// Mitsubishi GX Works2 project: Real Project Capstone   PLC: FX3U/FX3UC

PROGRAM MAIN
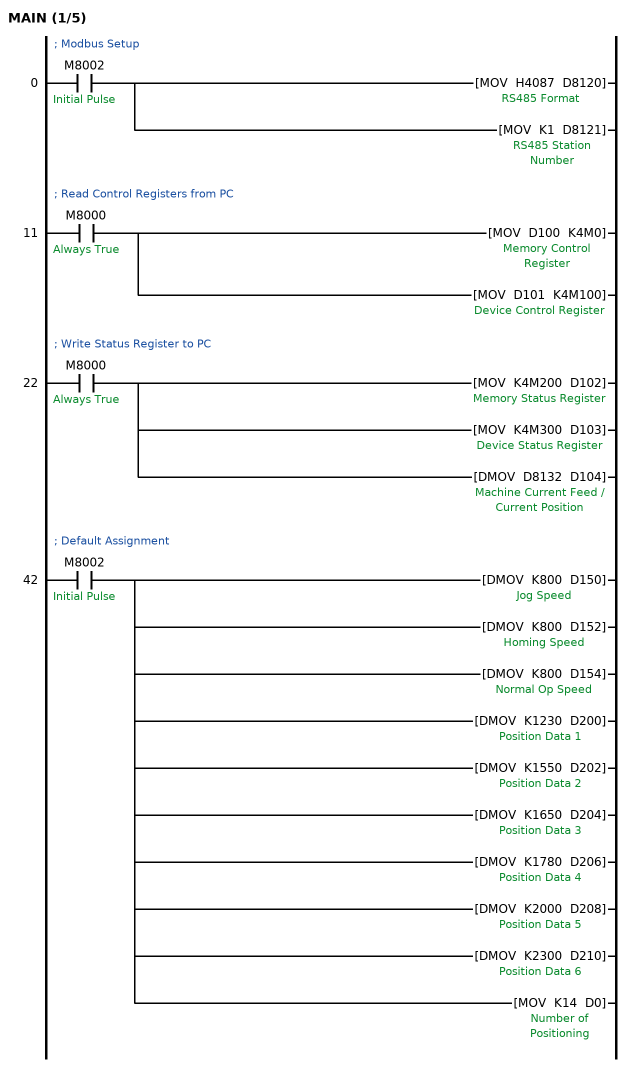
; Modbus Setup
0     LD      M8002  ; Initial Pulse
      MOV     H4087 D8120  ; RS485 Format
      MOV     K1 D8121  ; RS485 Station Number
; Read Control Registers from PC
11    LD      M8000  ; Always True
      MOV     D100 K4M0  ; Memory Control Register / Auto/Man Control
      MOV     D101 K4M100  ; Device Control Register / Light Control
; Write Status Register to PC
22    LD      M8000  ; Always True
      MOV     K4M200 D102  ; Start/Stop Status / Memory Status Register
      MOV     K4M300 D103  ; Light Status / Device Status Register
      DMOV    D8132 D104  ; Machine Current Feed / Current Position
; Default Assignment
42    LD      M8002  ; Initial Pulse
      DMOV    K800 D150  ; Jog Speed
      DMOV    K800 D152  ; Homing Speed
      DMOV    K800 D154  ; Normal Op Speed
      DMOV    K1230 D200  ; Position Data 1
      DMOV    K1550 D202  ; Position Data 2
      DMOV    K1650 D204  ; Position Data 3
      DMOV    K1780 D206  ; Position Data 4
      DMOV    K2000 D208  ; Position Data 5
      DMOV    K2300 D210  ; Position Data 6
      MOV     K14 D0  ; Number of Positioning
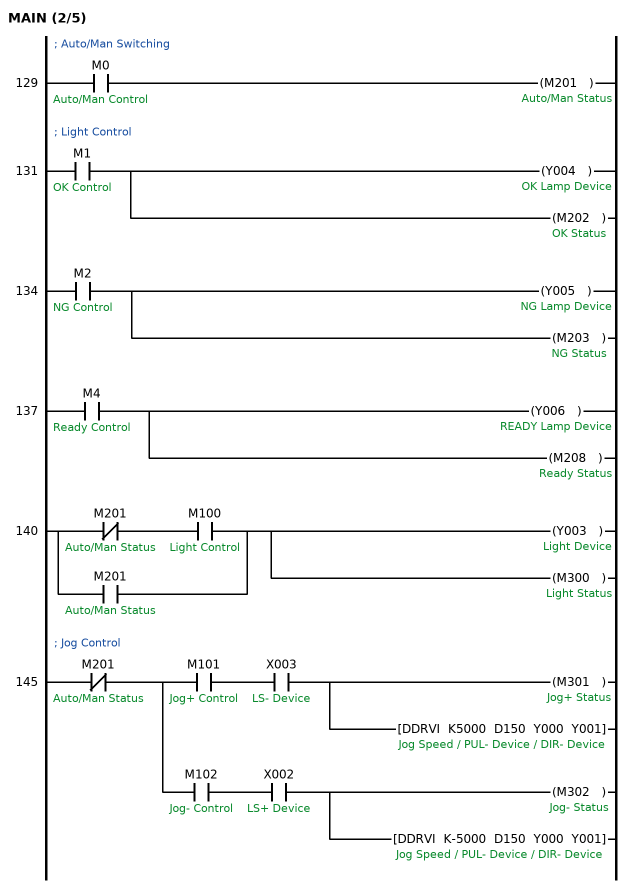
; Auto/Man Switching
129   LD      M0  ; Auto/Man Control
      OUT     M201  ; Auto/Man Status
; Light Control
131   LD      M1  ; OK Control
      OUT     Y004  ; OK Lamp Device
      OUT     M202  ; OK Status
134   LD      M2  ; NG Control
      OUT     Y005  ; NG Lamp Device
      OUT     M203  ; NG Status
137   LD      M4  ; Ready Control
      OUT     Y006  ; READY Lamp Device
      OUT     M208  ; Ready Status
140   LDI     M201  ; Auto/Man Status
      AND     M100  ; Light Control
      OR      M201  ; Auto/Man Status
      OUT     Y003  ; Light Device
      OUT     M300  ; Light Status
; Jog Control
145   LDI     M201  ; Auto/Man Status
      MPS
      AND     M101  ; Jog+ Control
      AND     X003  ; LS- Device
      OUT     M301  ; Jog+ Status
      DDRVI   K5000 D150 Y000 Y001  ; PUL- Device / DIR- Device
      MPP
      AND     M102  ; Jog- Control
      AND     X002  ; LS+ Device
      OUT     M302  ; Jog- Status
      DDRVI   K-5000 D150 Y000 Y001
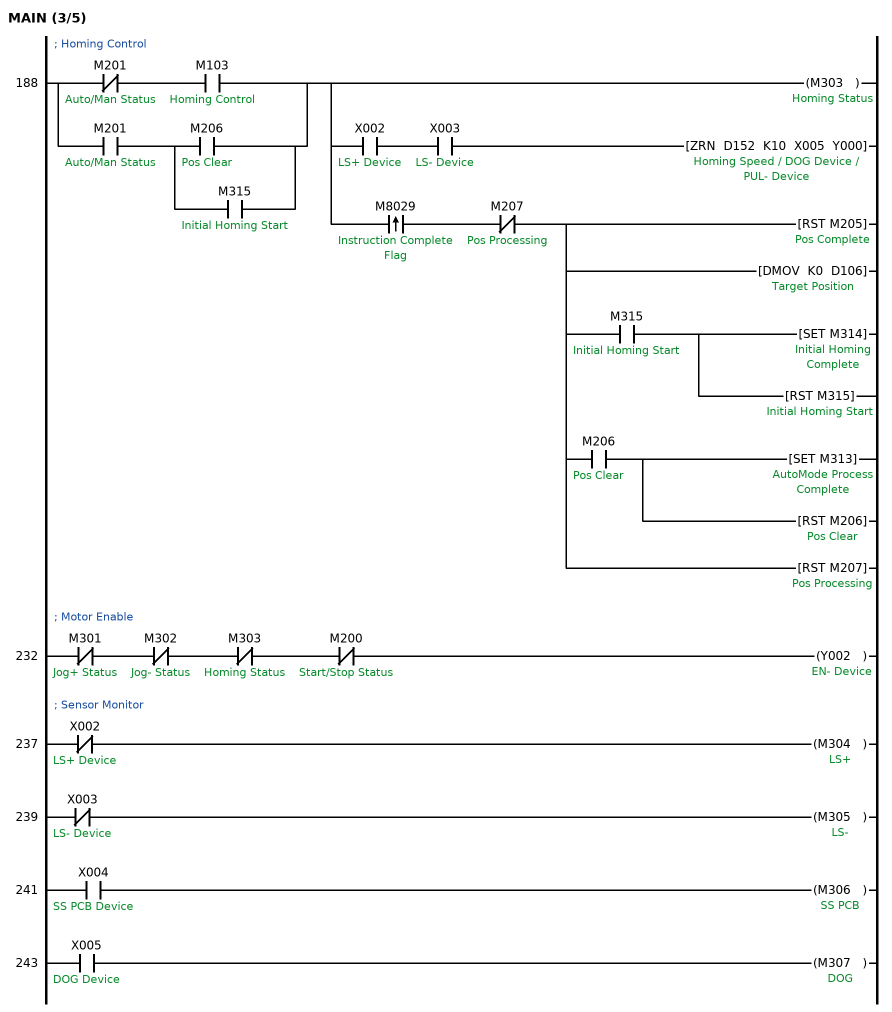
; Homing Control
188   LDI     M201  ; Auto/Man Status
      AND     M103  ; Homing Control
      LD      M201  ; Auto/Man Status
      LD      M206  ; Pos Clear
      OR      M315  ; Initial Homing Start
      ANB
      ORB
      OUT     M303  ; Homing Status
      MPS
      AND     X002  ; LS+ Device
      AND     X003  ; LS- Device
      ZRN     D152 K10 X005 Y000  ; DOG Device
      MPP
      ANDP    M8029  ; Instruction Complete Flag
      ANI     M207  ; Pos Processing
      RST     M205  ; Pos Complete
      DMOV    K0 D106  ; Target Position
      MPS
      AND     M315  ; Initial Homing Start
      SET     M314  ; Initial Homing Complete
      RST     M315  ; Initial Homing Start
      MRD
      AND     M206  ; Pos Clear
      SET     M313  ; AutoMode Process Complete
      RST     M206  ; Pos Clear
      MPP
      RST     M207  ; Pos Processing
; Motor Enable
232   LDI     M301  ; Jog+ Status
      ANI     M302  ; Jog- Status
      ANI     M303  ; Homing Status
      ANI     M200  ; Start/Stop Status
      OUT     Y002  ; EN- Device
; Sensor Monitor
237   LDI     X002  ; LS+ Device
      OUT     M304  ; LS+
239   LDI     X003  ; LS- Device
      OUT     M305  ; LS-
241   LD      X004  ; SS PCB Device
      OUT     M306  ; SS PCB
243   LD      X005  ; DOG Device
      OUT     M307  ; DOG
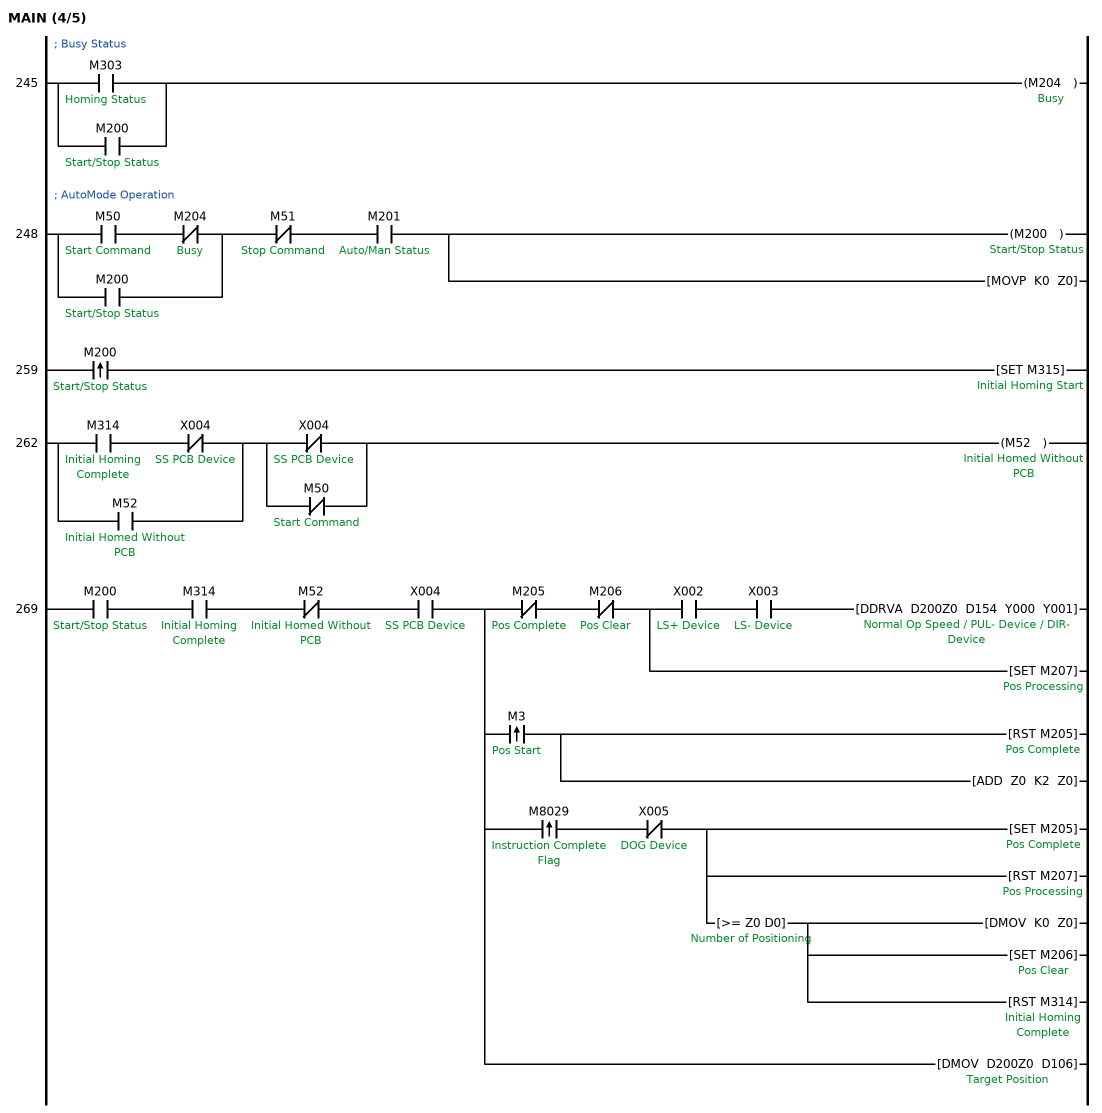
; Busy Status
245   LD      M303  ; Homing Status
      OR      M200  ; Start/Stop Status
      OUT     M204  ; Busy
; AutoMode Operation
248   LD      M50  ; Start Command
      ANI     M204  ; Busy
      OR      M200  ; Start/Stop Status
      ANI     M51  ; Stop Command
      AND     M201  ; Auto/Man Status
      OUT     M200  ; Start/Stop Status
      MOVP    K0 Z0
259   LDP     M200  ; Start/Stop Status
      SET     M315  ; Initial Homing Start
262   LD      M314  ; Initial Homing Complete
      ANI     X004  ; SS PCB Device
      OR      M52  ; Initial Homed Without PCB
      LDI     X004  ; SS PCB Device
      ORI     M50  ; Start Command
      ANB
      OUT     M52  ; Initial Homed Without PCB
269   LD      M200  ; Start/Stop Status
      AND     M314  ; Initial Homing Complete
      ANI     M52  ; Initial Homed Without PCB
      AND     X004  ; SS PCB Device
      MPS
      ANI     M205  ; Pos Complete
      ANI     M206  ; Pos Clear
      MPS
      AND     X002  ; LS+ Device
      AND     X003  ; LS- Device
      DDRVA   D200Z0 D154 Y000 Y001
      MPP
      SET     M207  ; Pos Processing
      MRD
      ANDP    M3  ; Pos Start
      RST     M205  ; Pos Complete
      ADD     Z0 K2 Z0
      MRD
      ANDP    M8029  ; Instruction Complete Flag
      ANI     X005  ; DOG Device
      SET     M205  ; Pos Complete
      RST     M207  ; Pos Processing
      AND>=   Z0 D0  ; Number of Positioning
      DMOV    K0 Z0
      SET     M206  ; Pos Clear
      RST     M314  ; Initial Homing Complete
      MPP
      DMOV    D200Z0 D106
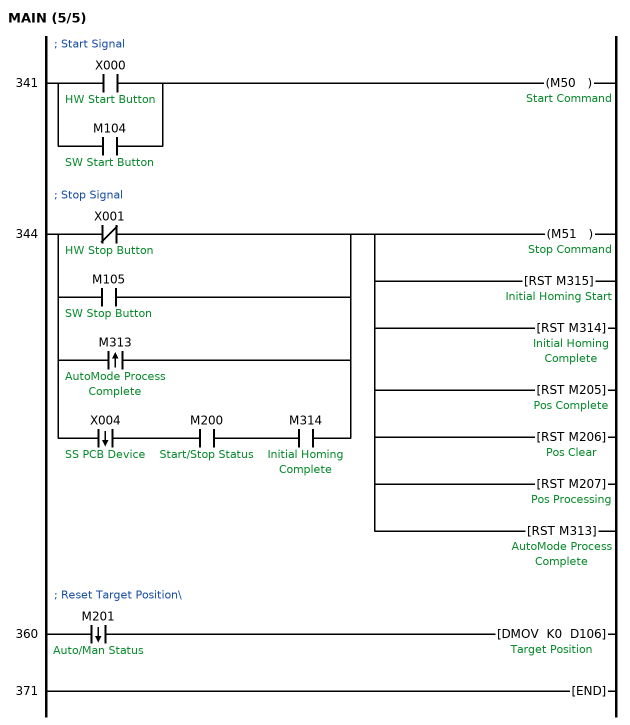
; Start Signal
341   LD      X000  ; HW Start Button
      OR      M104  ; SW Start Button
      OUT     M50  ; Start Command
; Stop Signal
344   LDI     X001  ; HW Stop Button
      OR      M105  ; SW Stop Button
      ORP     M313  ; AutoMode Process Complete
      LDF     X004  ; SS PCB Device
      AND     M200  ; Start/Stop Status
      AND     M314  ; Initial Homing Complete
      ORB
      OUT     M51  ; Stop Command
      RST     M315  ; Initial Homing Start
      RST     M314  ; Initial Homing Complete
      RST     M205  ; Pos Complete
      RST     M206  ; Pos Clear
      RST     M207  ; Pos Processing
      RST     M313  ; AutoMode Process Complete
; Reset Target Position\
360   LDF     M201  ; Auto/Man Status
      DMOV    K0 D106
371   END
END_PROGRAM

// device comments not shown above
M308  ; Forward
M309  ; Reversed
D212  ; Position Data 7
D214  ; Position Data 8
D216  ; Position Data 9
D218  ; Position Data 10
